// TIA Portal V16 export
// export: Created 2022-11-17T11:55:28.8325369Z, ExportSetting WithDefaults, DisplayName Totally Integrated Automation Portal, DisplayVersion V16 Update 6, DisplayName TIA Portal Version Control Interface, DisplayVersion V16 Update 2, DisplayName TIA Portal Openness, DisplayVersion V16 Update 6, DisplayName SINAMICS Startdrive Advanced, DisplayVersion V16 Update 5, DisplayName SINAMICS Startdrive G130, G150, S120, S150, SINAMICS MV, S210, DisplayVersion V16 Update 5, DisplayName SINAMICS Startdrive G110M, G120, G120C, G120D, G120P, G115D, DisplayVersion V16 Update 5, DisplayName STEP 7 Professional, DisplayVersion V16 Update 6, DisplayName STEP 7 Safety, DisplayVersion V16, DisplayName WinCC Advanced, DisplayVersion V16 Update 6
DATA_BLOCK "DB24_AlarmDisplay"   // DB24
{ S7_Optimized_Access := 'FALSE' }
AUTHOR : Robopac
VERSION : 0.0
// stored: AutoNumber false, IsOnlyStoredInLoadMemory false, IsWriteProtectedInAS false
   VAR RETAIN
      Alarm1 : Byte := 16#00;   // Alarm byte 1
      Alarm2 : Byte := 16#00;   // Alarm byte 2
      Alarm3 : Byte := 16#00;   // Alarm byte 3
      Alarm4 : Byte := 16#00;   // Alarm byte 4
      Alarm5 : Byte := 16#00;   // Alarm byte 5
      Alarm6 : Byte := 16#00;   // Alarm byte 6
      Alarm7 : Byte := 16#00;   // Alarm byte 7
      Alarm8 : Byte := 16#00;   // Alarm byte 8
      Alarm9 : Byte := 16#00;   // Alarm byte 9
      Alarm10 : Byte := 16#00;   // Alarm byte 10
      Alarm11 : Byte := 16#00;   // Alarm byte 11
      Alarm12 : Byte := 16#00;   // Alarm byte 12
      Alarm13 : Byte := 16#00;   // Alarm byte 13
      Alarm14 : Byte := 16#00;   // Alarm byte 14
      Alarm15 : Byte := 16#00;   // Alarm byte 15
      Alarm16 : Byte := 16#00;   // Alarm byte 16
      Alarm17 : Byte := 16#00;   // Alarm byte 17
      Alarm18 : Byte := 16#00;   // Alarm byte 18
      Alarm19 : Byte := 16#00;   // Alarm byte 19
      Alarm20 : Byte := 16#00;   // Alarm byte 20
      Alarm21 : Byte := 16#00;   // Alarm byte 21
      Alarm22 : Byte := 16#00;   // Alarm byte 22
      Alarm23 : Byte := 16#00;   // Alarm byte 23
      Alarm24 : Byte := 16#00;   // Alarm byte 24
      Alarm25 : Byte := 16#00;   // Alarm byte 25
      Alarm26 : Byte := 16#00;   // Alarm byte 26
      Alarm27 : Byte := 16#00;   // Alarm byte 27
      Alarm28 : Byte := 16#00;   // Alarm byte 28
      Alarm29 : Byte := 16#00;   // Alarm byte 29
      Alarm30 : Byte := 16#00;   // Alarm byte 30
      Alarm31 : Byte := 16#00;   // Alarm byte 31
      Alarm32 : Byte := 16#00;   // Alarm byte 32
      Alarm33 : Byte := 16#00;   // Alarm byte 33
      Alarm34 : Byte := 16#00;   // Alarm byte 34
      Alarm35 : Byte := 16#00;   // Alarm byte 35
      Alarm36 : Byte := 16#00;   // Alarm byte 36
      Alarm37 : Byte := 16#00;   // Alarm byte 37
      Alarm38 : Byte := 16#00;   // Alarm byte 38
      Alarm39 : Byte := 16#00;   // Alarm byte 39
      Alarm40 : Byte := 16#00;   // Alarm byte 40
      AckAlarm1 : Byte := 16#00;   // Alarm acknowledge for byte 1
      AckAlarm2 : Byte := 16#00;   // Alarm acknowledge for byte 2
      AckAlarm3 : Byte := 16#00;   // Alarm acknowledge for byte 3
      AckAlarm4 : Byte := 16#00;   // Alarm acknowledge for byte 4
      AckAlarm5 : Byte := 16#00;   // Alarm acknowledge for byte 5
      AckAlarm6 : Byte := 16#00;   // Alarm acknowledge for byte 6
      AckAlarm7 : Byte := 16#00;   // Alarm acknowledge for byte 7
      AckAlarm8 : Byte := 16#00;   // Alarm acknowledge for byte 8
      AckAlarm9 : Byte := 16#00;   // Alarm acknowledge for byte 9
      AckAlarm10 : Byte := 16#00;   // Alarm acknowledge for byte 10
      AckAlarm11 : Byte := 16#00;   // Alarm acknowledge for byte 11
      AckAlarm12 : Byte := 16#00;   // Alarm acknowledge for byte 12
      AckAlarm13 : Byte := 16#00;   // Alarm acknowledge for byte 13
      AckAlarm14 : Byte := 16#00;   // Alarm acknowledge for byte 14
      AckAlarm15 : Byte := 16#00;   // Alarm acknowledge for byte 15
      AckAlarm16 : Byte := 16#00;   // Alarm acknowledge for byte 16
      AckAlarm17 : Byte := 16#00;   // Alarm acknowledge for byte 17
      AckAlarm18 : Byte := 16#00;   // Alarm acknowledge for byte 18
      AckAlarm19 : Byte := 16#00;   // Alarm acknowledge for byte 19
      AckAlarm20 : Byte := 16#00;   // Alarm acknowledge for byte 20
      AckAlarm21 : Byte := 16#00;   // Alarm acknowledge for byte 21
      AckAlarm22 : Byte := 16#00;   // Alarm acknowledge for byte 22
      AckAlarm23 : Byte := 16#00;   // Alarm acknowledge for byte 23
      AckAlarm24 : Byte := 16#00;   // Alarm acknowledge for byte 24
      AckAlarm25 : Byte := 16#00;   // Alarm acknowledge for byte 25
      AckAlarm26 : Byte := 16#00;   // Alarm acknowledge for byte 26
      AckAlarm27 : Byte := 16#00;   // Alarm acknowledge for byte 27
      AckAlarm28 : Byte := 16#00;   // Alarm acknowledge for byte 28
      AckAlarm29 : Byte := 16#00;   // Alarm acknowledge for byte 29
      AckAlarm30 : Byte := 16#00;   // Alarm acknowledge for byte 30
      AckAlarm31 : Byte := 16#00;   // Alarm acknowledge for byte 31
      AckAlarm32 : Byte := 16#00;   // Alarm acknowledge for byte 32
      AckAlarm33 : Byte := 16#00;   // Alarm acknowledge for byte 33
      AckAlarm34 : Byte := 16#00;   // Alarm acknowledge for byte 34
      AckAlarm35 : Byte := 16#00;   // Alarm acknowledge for byte 35
      AckAlarm36 : Byte := 16#00;   // Alarm acknowledge for byte 36
      AckAlarm37 : Byte := 16#00;   // Alarm acknowledge for byte 37
      AckAlarm38 : Byte := 16#00;   // Alarm acknowledge for byte 38
      AckAlarm39 : Byte := 16#00;   // Alarm acknowledge for byte 39
      AckAlarm40 : Byte := 16#00;   // Alarm acknowledge for byte 40
   END_VAR
BEGIN
END_DATA_BLOCK
